TYPE TcoEntityBase EXTENDS TcoData.TcoEntity :
STRUCT
	{attribute clr [RenderIgnore("Control", "ShadowControl")]}
	{attribute addProperty Name "<#Created#>"}
	_Created : DT;
	{attribute clr [RenderIgnore("Control", "ShadowControl")]}
	{attribute addProperty Name "<#Modified#>"}
	_Modified : DT;
END_STRUCT
END_TYPE

(* stored: Version 1.1.0.1
   DUT TcoEntityBase: Id {82fa9cb5-c609-474c-9ff9-380ad63bb0af} *)
